FUNCTION_BLOCK FB60
TITLE = 'process_F1'
AUTHOR : CB

VAR
	tmp : BOOL;
END_VAR


BEGIN


NETWORK
TITLE =
//
//	process/process_F1/AscF1PROC
CALL FC59 (combE := 1);
CALL FB59,	DB59;
CALL FC59 (combE := 0);




END_FUNCTION_BLOCK
